// TIA Portal V16 export
// export: Created 2022-01-12T14:34:25.6760288Z, ExportSetting WithDefaults, DisplayName Totally Integrated Automation Portal, DisplayVersion V16 Update 4, DisplayName TIA Portal Version Control Interface, DisplayVersion V16 Update 2, DisplayName TIA Portal Openness, DisplayVersion V16 Update 4, DisplayName STEP 7 Professional, DisplayVersion V16 Update 4, DisplayName STEP 7 Safety, DisplayVersion V16, DisplayName WinCC Professional, DisplayVersion V16 Update 4
TYPE "typAlarmNew"
// stored: IsFailsafeCompliant false
   STRUCT
      stan : Int;   // 0-bark 1-wystapił i jest alarm
      procedura { ExternalAccessible := 'False'; ExternalVisible := 'False'; ExternalWritable := 'False'} : Int;   // numer procedury któa teraz wykonujemy
      timerek { ExternalAccessible := 'False'; ExternalVisible := 'False'; ExternalWritable := 'False'} : Int;   // czas liczony do wystapienia alarmu
   END_STRUCT;
END_TYPE
